TYPE "udtIOL-Hub"
VERSION : 0.1
   STRUCT
      "Byte" { ExternalAccessible := 'False'; ExternalVisible := 'False'; ExternalWritable := 'False'} : Array[0..1] of Byte;
   END_STRUCT;

END_TYPE

